Fanuc KAREL source: kt00454.compact.KL

PROGRAM KT00454
%STACKSIZE=65535
%PRIORITY=65535
%NOLOCKGROUP
VAR
H1 : ARRAY[2] OF SHORT
H2 : ARRAY[2] OF SHORT
OUT : BOOLEAN
BEGIN
H1[1]=2
H2[1]=3
H1[1]=2
H2[1]=3
OUT=(H1[1] >=H2[1])
END KT00454
